// TIA Portal V20 export
DATA_BLOCK "MotorStarterHMI"   // DB212
// stored: MemoryReserve 100
   VAR
      unitMotorstarter : Array[0.."NO_OF_UNITS"] of "typeEmMotorStarterInterface";
   END_VAR
BEGIN
   unitMotorstarter[0].EMmotorstarter[0].et200SpMotorstarterCurrent[0..1] := 0.0;
   unitMotorstarter[0].EMmotorstarter[1].et200SpMotorstarterCurrent[0..1] := 0.0;
   unitMotorstarter[0].EMmotorstarter[2].et200SpMotorstarterCurrent[0..1] := 0.0;
   unitMotorstarter[0].EMmotorstarter[3].et200SpMotorstarterCurrent[0..1] := 0.0;
   unitMotorstarter[0].EMmotorstarter[4].et200SpMotorstarterCurrent[0..1] := 0.0;
   unitMotorstarter[0].EMmotorstarter[5].et200SpMotorstarterCurrent[0..1] := 0.0;
   unitMotorstarter[0].EMmotorstarter[6].et200SpMotorstarterCurrent[0..1] := 0.0;
   unitMotorstarter[0].EMmotorstarter[7].et200SpMotorstarterCurrent[0..1] := 0.0;
   unitMotorstarter[0].EMmotorstarter[0].et200SpMotorstarterInputs[0..1].readyAutomatic := FALSE;
   unitMotorstarter[0].EMmotorstarter[1].et200SpMotorstarterInputs[0..1].readyAutomatic := FALSE;
   unitMotorstarter[0].EMmotorstarter[2].et200SpMotorstarterInputs[0..1].readyAutomatic := FALSE;
   unitMotorstarter[0].EMmotorstarter[3].et200SpMotorstarterInputs[0..1].readyAutomatic := FALSE;
   unitMotorstarter[0].EMmotorstarter[4].et200SpMotorstarterInputs[0..1].readyAutomatic := FALSE;
   unitMotorstarter[0].EMmotorstarter[5].et200SpMotorstarterInputs[0..1].readyAutomatic := FALSE;
   unitMotorstarter[0].EMmotorstarter[6].et200SpMotorstarterInputs[0..1].readyAutomatic := FALSE;
   unitMotorstarter[0].EMmotorstarter[7].et200SpMotorstarterInputs[0..1].readyAutomatic := FALSE;
   unitMotorstarter[0].EMmotorstarter[0].et200SpMotorstarterInputs[0..1].motorOn := FALSE;
   unitMotorstarter[0].EMmotorstarter[1].et200SpMotorstarterInputs[0..1].motorOn := FALSE;
   unitMotorstarter[0].EMmotorstarter[2].et200SpMotorstarterInputs[0..1].motorOn := FALSE;
   unitMotorstarter[0].EMmotorstarter[3].et200SpMotorstarterInputs[0..1].motorOn := FALSE;
   unitMotorstarter[0].EMmotorstarter[4].et200SpMotorstarterInputs[0..1].motorOn := FALSE;
   unitMotorstarter[0].EMmotorstarter[5].et200SpMotorstarterInputs[0..1].motorOn := FALSE;
   unitMotorstarter[0].EMmotorstarter[6].et200SpMotorstarterInputs[0..1].motorOn := FALSE;
   unitMotorstarter[0].EMmotorstarter[7].et200SpMotorstarterInputs[0..1].motorOn := FALSE;
   unitMotorstarter[0].EMmotorstarter[0].et200SpMotorstarterInputs[0..1].groupFault := FALSE;
   unitMotorstarter[0].EMmotorstarter[1].et200SpMotorstarterInputs[0..1].groupFault := FALSE;
   unitMotorstarter[0].EMmotorstarter[2].et200SpMotorstarterInputs[0..1].groupFault := FALSE;
   unitMotorstarter[0].EMmotorstarter[3].et200SpMotorstarterInputs[0..1].groupFault := FALSE;
   unitMotorstarter[0].EMmotorstarter[4].et200SpMotorstarterInputs[0..1].groupFault := FALSE;
   unitMotorstarter[0].EMmotorstarter[5].et200SpMotorstarterInputs[0..1].groupFault := FALSE;
   unitMotorstarter[0].EMmotorstarter[6].et200SpMotorstarterInputs[0..1].groupFault := FALSE;
   unitMotorstarter[0].EMmotorstarter[7].et200SpMotorstarterInputs[0..1].groupFault := FALSE;
   unitMotorstarter[0].EMmotorstarter[0].et200SpMotorstarterInputs[0..1].groupWarning := FALSE;
   unitMotorstarter[0].EMmotorstarter[1].et200SpMotorstarterInputs[0..1].groupWarning := FALSE;
   unitMotorstarter[0].EMmotorstarter[2].et200SpMotorstarterInputs[0..1].groupWarning := FALSE;
   unitMotorstarter[0].EMmotorstarter[3].et200SpMotorstarterInputs[0..1].groupWarning := FALSE;
   unitMotorstarter[0].EMmotorstarter[4].et200SpMotorstarterInputs[0..1].groupWarning := FALSE;
   unitMotorstarter[0].EMmotorstarter[5].et200SpMotorstarterInputs[0..1].groupWarning := FALSE;
   unitMotorstarter[0].EMmotorstarter[6].et200SpMotorstarterInputs[0..1].groupWarning := FALSE;
   unitMotorstarter[0].EMmotorstarter[7].et200SpMotorstarterInputs[0..1].groupWarning := FALSE;
   unitMotorstarter[0].EMmotorstarter[0].et200SpMotorstarterInputs[0..1].input1 := FALSE;
   unitMotorstarter[0].EMmotorstarter[1].et200SpMotorstarterInputs[0..1].input1 := FALSE;
   unitMotorstarter[0].EMmotorstarter[2].et200SpMotorstarterInputs[0..1].input1 := FALSE;
   unitMotorstarter[0].EMmotorstarter[3].et200SpMotorstarterInputs[0..1].input1 := FALSE;
   unitMotorstarter[0].EMmotorstarter[4].et200SpMotorstarterInputs[0..1].input1 := FALSE;
   unitMotorstarter[0].EMmotorstarter[5].et200SpMotorstarterInputs[0..1].input1 := FALSE;
   unitMotorstarter[0].EMmotorstarter[6].et200SpMotorstarterInputs[0..1].input1 := FALSE;
   unitMotorstarter[0].EMmotorstarter[7].et200SpMotorstarterInputs[0..1].input1 := FALSE;
   unitMotorstarter[0].EMmotorstarter[0].et200SpMotorstarterInputs[0..1].input2 := FALSE;
   unitMotorstarter[0].EMmotorstarter[1].et200SpMotorstarterInputs[0..1].input2 := FALSE;
   unitMotorstarter[0].EMmotorstarter[2].et200SpMotorstarterInputs[0..1].input2 := FALSE;
   unitMotorstarter[0].EMmotorstarter[3].et200SpMotorstarterInputs[0..1].input2 := FALSE;
   unitMotorstarter[0].EMmotorstarter[4].et200SpMotorstarterInputs[0..1].input2 := FALSE;
   unitMotorstarter[0].EMmotorstarter[5].et200SpMotorstarterInputs[0..1].input2 := FALSE;
   unitMotorstarter[0].EMmotorstarter[6].et200SpMotorstarterInputs[0..1].input2 := FALSE;
   unitMotorstarter[0].EMmotorstarter[7].et200SpMotorstarterInputs[0..1].input2 := FALSE;
   unitMotorstarter[0].EMmotorstarter[0].et200SpMotorstarterInputs[0..1].input3 := FALSE;
   unitMotorstarter[0].EMmotorstarter[1].et200SpMotorstarterInputs[0..1].input3 := FALSE;
   unitMotorstarter[0].EMmotorstarter[2].et200SpMotorstarterInputs[0..1].input3 := FALSE;
   unitMotorstarter[0].EMmotorstarter[3].et200SpMotorstarterInputs[0..1].input3 := FALSE;
   unitMotorstarter[0].EMmotorstarter[4].et200SpMotorstarterInputs[0..1].input3 := FALSE;
   unitMotorstarter[0].EMmotorstarter[5].et200SpMotorstarterInputs[0..1].input3 := FALSE;
   unitMotorstarter[0].EMmotorstarter[6].et200SpMotorstarterInputs[0..1].input3 := FALSE;
   unitMotorstarter[0].EMmotorstarter[7].et200SpMotorstarterInputs[0..1].input3 := FALSE;
   unitMotorstarter[0].EMmotorstarter[0].et200SpMotorstarterInputs[0..1].inputLocalCtrl := FALSE;
   unitMotorstarter[0].EMmotorstarter[1].et200SpMotorstarterInputs[0..1].inputLocalCtrl := FALSE;
   unitMotorstarter[0].EMmotorstarter[2].et200SpMotorstarterInputs[0..1].inputLocalCtrl := FALSE;
   unitMotorstarter[0].EMmotorstarter[3].et200SpMotorstarterInputs[0..1].inputLocalCtrl := FALSE;
   unitMotorstarter[0].EMmotorstarter[4].et200SpMotorstarterInputs[0..1].inputLocalCtrl := FALSE;
   unitMotorstarter[0].EMmotorstarter[5].et200SpMotorstarterInputs[0..1].inputLocalCtrl := FALSE;
   unitMotorstarter[0].EMmotorstarter[6].et200SpMotorstarterInputs[0..1].inputLocalCtrl := FALSE;
   unitMotorstarter[0].EMmotorstarter[7].et200SpMotorstarterInputs[0..1].inputLocalCtrl := FALSE;
   unitMotorstarter[0].EMmotorstarter[0].et200SpMotorstarterInputs[0..1].iActBit0 := FALSE;
   unitMotorstarter[0].EMmotorstarter[1].et200SpMotorstarterInputs[0..1].iActBit0 := FALSE;
   unitMotorstarter[0].EMmotorstarter[2].et200SpMotorstarterInputs[0..1].iActBit0 := FALSE;
   unitMotorstarter[0].EMmotorstarter[3].et200SpMotorstarterInputs[0..1].iActBit0 := FALSE;
   unitMotorstarter[0].EMmotorstarter[4].et200SpMotorstarterInputs[0..1].iActBit0 := FALSE;
   unitMotorstarter[0].EMmotorstarter[5].et200SpMotorstarterInputs[0..1].iActBit0 := FALSE;
   unitMotorstarter[0].EMmotorstarter[6].et200SpMotorstarterInputs[0..1].iActBit0 := FALSE;
   unitMotorstarter[0].EMmotorstarter[7].et200SpMotorstarterInputs[0..1].iActBit0 := FALSE;
   unitMotorstarter[0].EMmotorstarter[0].et200SpMotorstarterInputs[0..1].iActBit1 := FALSE;
   unitMotorstarter[0].EMmotorstarter[1].et200SpMotorstarterInputs[0..1].iActBit1 := FALSE;
   unitMotorstarter[0].EMmotorstarter[2].et200SpMotorstarterInputs[0..1].iActBit1 := FALSE;
   unitMotorstarter[0].EMmotorstarter[3].et200SpMotorstarterInputs[0..1].iActBit1 := FALSE;
   unitMotorstarter[0].EMmotorstarter[4].et200SpMotorstarterInputs[0..1].iActBit1 := FALSE;
   unitMotorstarter[0].EMmotorstarter[5].et200SpMotorstarterInputs[0..1].iActBit1 := FALSE;
   unitMotorstarter[0].EMmotorstarter[6].et200SpMotorstarterInputs[0..1].iActBit1 := FALSE;
   unitMotorstarter[0].EMmotorstarter[7].et200SpMotorstarterInputs[0..1].iActBit1 := FALSE;
   unitMotorstarter[0].EMmotorstarter[0].et200SpMotorstarterInputs[0..1].iActBit2 := FALSE;
   unitMotorstarter[0].EMmotorstarter[1].et200SpMotorstarterInputs[0..1].iActBit2 := FALSE;
   unitMotorstarter[0].EMmotorstarter[2].et200SpMotorstarterInputs[0..1].iActBit2 := FALSE;
   unitMotorstarter[0].EMmotorstarter[3].et200SpMotorstarterInputs[0..1].iActBit2 := FALSE;
   unitMotorstarter[0].EMmotorstarter[4].et200SpMotorstarterInputs[0..1].iActBit2 := FALSE;
   unitMotorstarter[0].EMmotorstarter[5].et200SpMotorstarterInputs[0..1].iActBit2 := FALSE;
   unitMotorstarter[0].EMmotorstarter[6].et200SpMotorstarterInputs[0..1].iActBit2 := FALSE;
   unitMotorstarter[0].EMmotorstarter[7].et200SpMotorstarterInputs[0..1].iActBit2 := FALSE;
   unitMotorstarter[0].EMmotorstarter[0].et200SpMotorstarterInputs[0..1].iActBit3 := FALSE;
   unitMotorstarter[0].EMmotorstarter[1].et200SpMotorstarterInputs[0..1].iActBit3 := FALSE;
   unitMotorstarter[0].EMmotorstarter[2].et200SpMotorstarterInputs[0..1].iActBit3 := FALSE;
   unitMotorstarter[0].EMmotorstarter[3].et200SpMotorstarterInputs[0..1].iActBit3 := FALSE;
   unitMotorstarter[0].EMmotorstarter[4].et200SpMotorstarterInputs[0..1].iActBit3 := FALSE;
   unitMotorstarter[0].EMmotorstarter[5].et200SpMotorstarterInputs[0..1].iActBit3 := FALSE;
   unitMotorstarter[0].EMmotorstarter[6].et200SpMotorstarterInputs[0..1].iActBit3 := FALSE;
   unitMotorstarter[0].EMmotorstarter[7].et200SpMotorstarterInputs[0..1].iActBit3 := FALSE;
   unitMotorstarter[0].EMmotorstarter[0].et200SpMotorstarterInputs[0..1].iActBit4 := FALSE;
   unitMotorstarter[0].EMmotorstarter[1].et200SpMotorstarterInputs[0..1].iActBit4 := FALSE;
   unitMotorstarter[0].EMmotorstarter[2].et200SpMotorstarterInputs[0..1].iActBit4 := FALSE;
   unitMotorstarter[0].EMmotorstarter[3].et200SpMotorstarterInputs[0..1].iActBit4 := FALSE;
   unitMotorstarter[0].EMmotorstarter[4].et200SpMotorstarterInputs[0..1].iActBit4 := FALSE;
   unitMotorstarter[0].EMmotorstarter[5].et200SpMotorstarterInputs[0..1].iActBit4 := FALSE;
   unitMotorstarter[0].EMmotorstarter[6].et200SpMotorstarterInputs[0..1].iActBit4 := FALSE;
   unitMotorstarter[0].EMmotorstarter[7].et200SpMotorstarterInputs[0..1].iActBit4 := FALSE;
   unitMotorstarter[0].EMmotorstarter[0].et200SpMotorstarterInputs[0..1].iActBit5 := FALSE;
   unitMotorstarter[0].EMmotorstarter[1].et200SpMotorstarterInputs[0..1].iActBit5 := FALSE;
   unitMotorstarter[0].EMmotorstarter[2].et200SpMotorstarterInputs[0..1].iActBit5 := FALSE;
   unitMotorstarter[0].EMmotorstarter[3].et200SpMotorstarterInputs[0..1].iActBit5 := FALSE;
   unitMotorstarter[0].EMmotorstarter[4].et200SpMotorstarterInputs[0..1].iActBit5 := FALSE;
   unitMotorstarter[0].EMmotorstarter[5].et200SpMotorstarterInputs[0..1].iActBit5 := FALSE;
   unitMotorstarter[0].EMmotorstarter[6].et200SpMotorstarterInputs[0..1].iActBit5 := FALSE;
   unitMotorstarter[0].EMmotorstarter[7].et200SpMotorstarterInputs[0..1].iActBit5 := FALSE;
   unitMotorstarter[0].EMmotorstarter[0].et200SpMotorstarterInputs[0..1].manualOperating := FALSE;
   unitMotorstarter[0].EMmotorstarter[1].et200SpMotorstarterInputs[0..1].manualOperating := FALSE;
   unitMotorstarter[0].EMmotorstarter[2].et200SpMotorstarterInputs[0..1].manualOperating := FALSE;
   unitMotorstarter[0].EMmotorstarter[3].et200SpMotorstarterInputs[0..1].manualOperating := FALSE;
   unitMotorstarter[0].EMmotorstarter[4].et200SpMotorstarterInputs[0..1].manualOperating := FALSE;
   unitMotorstarter[0].EMmotorstarter[5].et200SpMotorstarterInputs[0..1].manualOperating := FALSE;
   unitMotorstarter[0].EMmotorstarter[6].et200SpMotorstarterInputs[0..1].manualOperating := FALSE;
   unitMotorstarter[0].EMmotorstarter[7].et200SpMotorstarterInputs[0..1].manualOperating := FALSE;
   unitMotorstarter[0].EMmotorstarter[0].et200SpMotorstarterInputs[0..1].spare1 := FALSE;
   unitMotorstarter[0].EMmotorstarter[1].et200SpMotorstarterInputs[0..1].spare1 := FALSE;
   unitMotorstarter[0].EMmotorstarter[2].et200SpMotorstarterInputs[0..1].spare1 := FALSE;
   unitMotorstarter[0].EMmotorstarter[3].et200SpMotorstarterInputs[0..1].spare1 := FALSE;
   unitMotorstarter[0].EMmotorstarter[4].et200SpMotorstarterInputs[0..1].spare1 := FALSE;
   unitMotorstarter[0].EMmotorstarter[5].et200SpMotorstarterInputs[0..1].spare1 := FALSE;
   unitMotorstarter[0].EMmotorstarter[6].et200SpMotorstarterInputs[0..1].spare1 := FALSE;
   unitMotorstarter[0].EMmotorstarter[7].et200SpMotorstarterInputs[0..1].spare1 := FALSE;
   unitMotorstarter[0].EMmotorstarter[0].et200SpMotorstarterInputs[0..1].readyStartOn := FALSE;
   unitMotorstarter[0].EMmotorstarter[1].et200SpMotorstarterInputs[0..1].readyStartOn := FALSE;
   unitMotorstarter[0].EMmotorstarter[2].et200SpMotorstarterInputs[0..1].readyStartOn := FALSE;
   unitMotorstarter[0].EMmotorstarter[3].et200SpMotorstarterInputs[0..1].readyStartOn := FALSE;
   unitMotorstarter[0].EMmotorstarter[4].et200SpMotorstarterInputs[0..1].readyStartOn := FALSE;
   unitMotorstarter[0].EMmotorstarter[5].et200SpMotorstarterInputs[0..1].readyStartOn := FALSE;
   unitMotorstarter[0].EMmotorstarter[6].et200SpMotorstarterInputs[0..1].readyStartOn := FALSE;
   unitMotorstarter[0].EMmotorstarter[7].et200SpMotorstarterInputs[0..1].readyStartOn := FALSE;
   unitMotorstarter[0].EMmotorstarter[0].et200SpMotorstarterInputs[0..1].motorOnRight := FALSE;
   unitMotorstarter[0].EMmotorstarter[1].et200SpMotorstarterInputs[0..1].motorOnRight := FALSE;
   unitMotorstarter[0].EMmotorstarter[2].et200SpMotorstarterInputs[0..1].motorOnRight := FALSE;
   unitMotorstarter[0].EMmotorstarter[3].et200SpMotorstarterInputs[0..1].motorOnRight := FALSE;
   unitMotorstarter[0].EMmotorstarter[4].et200SpMotorstarterInputs[0..1].motorOnRight := FALSE;
   unitMotorstarter[0].EMmotorstarter[5].et200SpMotorstarterInputs[0..1].motorOnRight := FALSE;
   unitMotorstarter[0].EMmotorstarter[6].et200SpMotorstarterInputs[0..1].motorOnRight := FALSE;
   unitMotorstarter[0].EMmotorstarter[7].et200SpMotorstarterInputs[0..1].motorOnRight := FALSE;
   unitMotorstarter[0].EMmotorstarter[0].et200SpMotorstarterInputs[0..1].motorOnLeft := FALSE;
   unitMotorstarter[0].EMmotorstarter[1].et200SpMotorstarterInputs[0..1].motorOnLeft := FALSE;
   unitMotorstarter[0].EMmotorstarter[2].et200SpMotorstarterInputs[0..1].motorOnLeft := FALSE;
   unitMotorstarter[0].EMmotorstarter[3].et200SpMotorstarterInputs[0..1].motorOnLeft := FALSE;
   unitMotorstarter[0].EMmotorstarter[4].et200SpMotorstarterInputs[0..1].motorOnLeft := FALSE;
   unitMotorstarter[0].EMmotorstarter[5].et200SpMotorstarterInputs[0..1].motorOnLeft := FALSE;
   unitMotorstarter[0].EMmotorstarter[6].et200SpMotorstarterInputs[0..1].motorOnLeft := FALSE;
   unitMotorstarter[0].EMmotorstarter[7].et200SpMotorstarterInputs[0..1].motorOnLeft := FALSE;
   unitMotorstarter[0].EMmotorstarter[0].et200SpMotorstarterInputs[0..1].quickstopActive := FALSE;
   unitMotorstarter[0].EMmotorstarter[1].et200SpMotorstarterInputs[0..1].quickstopActive := FALSE;
   unitMotorstarter[0].EMmotorstarter[2].et200SpMotorstarterInputs[0..1].quickstopActive := FALSE;
   unitMotorstarter[0].EMmotorstarter[3].et200SpMotorstarterInputs[0..1].quickstopActive := FALSE;
   unitMotorstarter[0].EMmotorstarter[4].et200SpMotorstarterInputs[0..1].quickstopActive := FALSE;
   unitMotorstarter[0].EMmotorstarter[5].et200SpMotorstarterInputs[0..1].quickstopActive := FALSE;
   unitMotorstarter[0].EMmotorstarter[6].et200SpMotorstarterInputs[0..1].quickstopActive := FALSE;
   unitMotorstarter[0].EMmotorstarter[7].et200SpMotorstarterInputs[0..1].quickstopActive := FALSE;
   unitMotorstarter[0].EMmotorstarter[0].et200SpMotorstarterInputs[0..1].energySaving := FALSE;
   unitMotorstarter[0].EMmotorstarter[1].et200SpMotorstarterInputs[0..1].energySaving := FALSE;
   unitMotorstarter[0].EMmotorstarter[2].et200SpMotorstarterInputs[0..1].energySaving := FALSE;
   unitMotorstarter[0].EMmotorstarter[3].et200SpMotorstarterInputs[0..1].energySaving := FALSE;
   unitMotorstarter[0].EMmotorstarter[4].et200SpMotorstarterInputs[0..1].energySaving := FALSE;
   unitMotorstarter[0].EMmotorstarter[5].et200SpMotorstarterInputs[0..1].energySaving := FALSE;
   unitMotorstarter[0].EMmotorstarter[6].et200SpMotorstarterInputs[0..1].energySaving := FALSE;
   unitMotorstarter[0].EMmotorstarter[7].et200SpMotorstarterInputs[0..1].energySaving := FALSE;
   unitMotorstarter[0].EMmotorstarter[0].et200SpMotorstarterInputs[0..1].moduleInserted := FALSE;
   unitMotorstarter[0].EMmotorstarter[1].et200SpMotorstarterInputs[0..1].moduleInserted := FALSE;
   unitMotorstarter[0].EMmotorstarter[2].et200SpMotorstarterInputs[0..1].moduleInserted := FALSE;
   unitMotorstarter[0].EMmotorstarter[3].et200SpMotorstarterInputs[0..1].moduleInserted := FALSE;
   unitMotorstarter[0].EMmotorstarter[4].et200SpMotorstarterInputs[0..1].moduleInserted := FALSE;
   unitMotorstarter[0].EMmotorstarter[5].et200SpMotorstarterInputs[0..1].moduleInserted := FALSE;
   unitMotorstarter[0].EMmotorstarter[6].et200SpMotorstarterInputs[0..1].moduleInserted := FALSE;
   unitMotorstarter[0].EMmotorstarter[7].et200SpMotorstarterInputs[0..1].moduleInserted := FALSE;
   unitMotorstarter[0].EMmotorstarter[0].et200SpMotorstarterInputs[0..1].exProtectionMotorActive := FALSE;
   unitMotorstarter[0].EMmotorstarter[1].et200SpMotorstarterInputs[0..1].exProtectionMotorActive := FALSE;
   unitMotorstarter[0].EMmotorstarter[2].et200SpMotorstarterInputs[0..1].exProtectionMotorActive := FALSE;
   unitMotorstarter[0].EMmotorstarter[3].et200SpMotorstarterInputs[0..1].exProtectionMotorActive := FALSE;
   unitMotorstarter[0].EMmotorstarter[4].et200SpMotorstarterInputs[0..1].exProtectionMotorActive := FALSE;
   unitMotorstarter[0].EMmotorstarter[5].et200SpMotorstarterInputs[0..1].exProtectionMotorActive := FALSE;
   unitMotorstarter[0].EMmotorstarter[6].et200SpMotorstarterInputs[0..1].exProtectionMotorActive := FALSE;
   unitMotorstarter[0].EMmotorstarter[7].et200SpMotorstarterInputs[0..1].exProtectionMotorActive := FALSE;
   unitMotorstarter[0].EMmotorstarter[0].et200SpMotorstarterInputs[0..1].blockActive := FALSE;
   unitMotorstarter[0].EMmotorstarter[1].et200SpMotorstarterInputs[0..1].blockActive := FALSE;
   unitMotorstarter[0].EMmotorstarter[2].et200SpMotorstarterInputs[0..1].blockActive := FALSE;
   unitMotorstarter[0].EMmotorstarter[3].et200SpMotorstarterInputs[0..1].blockActive := FALSE;
   unitMotorstarter[0].EMmotorstarter[4].et200SpMotorstarterInputs[0..1].blockActive := FALSE;
   unitMotorstarter[0].EMmotorstarter[5].et200SpMotorstarterInputs[0..1].blockActive := FALSE;
   unitMotorstarter[0].EMmotorstarter[6].et200SpMotorstarterInputs[0..1].blockActive := FALSE;
   unitMotorstarter[0].EMmotorstarter[7].et200SpMotorstarterInputs[0..1].blockActive := FALSE;
   unitMotorstarter[0].EMmotorstarter[0].et200SpMotorstarterInputs[0..1].thermalMotorOverload := FALSE;
   unitMotorstarter[0].EMmotorstarter[1].et200SpMotorstarterInputs[0..1].thermalMotorOverload := FALSE;
   unitMotorstarter[0].EMmotorstarter[2].et200SpMotorstarterInputs[0..1].thermalMotorOverload := FALSE;
   unitMotorstarter[0].EMmotorstarter[3].et200SpMotorstarterInputs[0..1].thermalMotorOverload := FALSE;
   unitMotorstarter[0].EMmotorstarter[4].et200SpMotorstarterInputs[0..1].thermalMotorOverload := FALSE;
   unitMotorstarter[0].EMmotorstarter[5].et200SpMotorstarterInputs[0..1].thermalMotorOverload := FALSE;
   unitMotorstarter[0].EMmotorstarter[6].et200SpMotorstarterInputs[0..1].thermalMotorOverload := FALSE;
   unitMotorstarter[0].EMmotorstarter[7].et200SpMotorstarterInputs[0..1].thermalMotorOverload := FALSE;
   unitMotorstarter[0].EMmotorstarter[0].et200SpMotorstarterInputs[0..1].spare5 := FALSE;
   unitMotorstarter[0].EMmotorstarter[1].et200SpMotorstarterInputs[0..1].spare5 := FALSE;
   unitMotorstarter[0].EMmotorstarter[2].et200SpMotorstarterInputs[0..1].spare5 := FALSE;
   unitMotorstarter[0].EMmotorstarter[3].et200SpMotorstarterInputs[0..1].spare5 := FALSE;
   unitMotorstarter[0].EMmotorstarter[4].et200SpMotorstarterInputs[0..1].spare5 := FALSE;
   unitMotorstarter[0].EMmotorstarter[5].et200SpMotorstarterInputs[0..1].spare5 := FALSE;
   unitMotorstarter[0].EMmotorstarter[6].et200SpMotorstarterInputs[0..1].spare5 := FALSE;
   unitMotorstarter[0].EMmotorstarter[7].et200SpMotorstarterInputs[0..1].spare5 := FALSE;
   unitMotorstarter[0].EMmotorstarter[0].et200SpMotorstarterInputs[0..1].currentLimitTripping := FALSE;
   unitMotorstarter[0].EMmotorstarter[1].et200SpMotorstarterInputs[0..1].currentLimitTripping := FALSE;
   unitMotorstarter[0].EMmotorstarter[2].et200SpMotorstarterInputs[0..1].currentLimitTripping := FALSE;
   unitMotorstarter[0].EMmotorstarter[3].et200SpMotorstarterInputs[0..1].currentLimitTripping := FALSE;
   unitMotorstarter[0].EMmotorstarter[4].et200SpMotorstarterInputs[0..1].currentLimitTripping := FALSE;
   unitMotorstarter[0].EMmotorstarter[5].et200SpMotorstarterInputs[0..1].currentLimitTripping := FALSE;
   unitMotorstarter[0].EMmotorstarter[6].et200SpMotorstarterInputs[0..1].currentLimitTripping := FALSE;
   unitMotorstarter[0].EMmotorstarter[7].et200SpMotorstarterInputs[0..1].currentLimitTripping := FALSE;
   unitMotorstarter[0].EMmotorstarter[0].et200SpMotorstarterInputs[0..1].statusFailDi := FALSE;
   unitMotorstarter[0].EMmotorstarter[1].et200SpMotorstarterInputs[0..1].statusFailDi := FALSE;
   unitMotorstarter[0].EMmotorstarter[2].et200SpMotorstarterInputs[0..1].statusFailDi := FALSE;
   unitMotorstarter[0].EMmotorstarter[3].et200SpMotorstarterInputs[0..1].statusFailDi := FALSE;
   unitMotorstarter[0].EMmotorstarter[4].et200SpMotorstarterInputs[0..1].statusFailDi := FALSE;
   unitMotorstarter[0].EMmotorstarter[5].et200SpMotorstarterInputs[0..1].statusFailDi := FALSE;
   unitMotorstarter[0].EMmotorstarter[6].et200SpMotorstarterInputs[0..1].statusFailDi := FALSE;
   unitMotorstarter[0].EMmotorstarter[7].et200SpMotorstarterInputs[0..1].statusFailDi := FALSE;
   unitMotorstarter[0].EMmotorstarter[0].et200SpMotorstarterInputs[0..1].residualCurrent := FALSE;
   unitMotorstarter[0].EMmotorstarter[1].et200SpMotorstarterInputs[0..1].residualCurrent := FALSE;
   unitMotorstarter[0].EMmotorstarter[2].et200SpMotorstarterInputs[0..1].residualCurrent := FALSE;
   unitMotorstarter[0].EMmotorstarter[3].et200SpMotorstarterInputs[0..1].residualCurrent := FALSE;
   unitMotorstarter[0].EMmotorstarter[4].et200SpMotorstarterInputs[0..1].residualCurrent := FALSE;
   unitMotorstarter[0].EMmotorstarter[5].et200SpMotorstarterInputs[0..1].residualCurrent := FALSE;
   unitMotorstarter[0].EMmotorstarter[6].et200SpMotorstarterInputs[0..1].residualCurrent := FALSE;
   unitMotorstarter[0].EMmotorstarter[7].et200SpMotorstarterInputs[0..1].residualCurrent := FALSE;
   unitMotorstarter[0].EMmotorstarter[0].et200SpMotorstarterInputs[0..1].asymmetryDetected := FALSE;
   unitMotorstarter[0].EMmotorstarter[1].et200SpMotorstarterInputs[0..1].asymmetryDetected := FALSE;
   unitMotorstarter[0].EMmotorstarter[2].et200SpMotorstarterInputs[0..1].asymmetryDetected := FALSE;
   unitMotorstarter[0].EMmotorstarter[3].et200SpMotorstarterInputs[0..1].asymmetryDetected := FALSE;
   unitMotorstarter[0].EMmotorstarter[4].et200SpMotorstarterInputs[0..1].asymmetryDetected := FALSE;
   unitMotorstarter[0].EMmotorstarter[5].et200SpMotorstarterInputs[0..1].asymmetryDetected := FALSE;
   unitMotorstarter[0].EMmotorstarter[6].et200SpMotorstarterInputs[0..1].asymmetryDetected := FALSE;
   unitMotorstarter[0].EMmotorstarter[7].et200SpMotorstarterInputs[0..1].asymmetryDetected := FALSE;
   unitMotorstarter[0].EMmotorstarter[0].et200SpMotorstarterInputs[0..1].overtemperature := FALSE;
   unitMotorstarter[0].EMmotorstarter[1].et200SpMotorstarterInputs[0..1].overtemperature := FALSE;
   unitMotorstarter[0].EMmotorstarter[2].et200SpMotorstarterInputs[0..1].overtemperature := FALSE;
   unitMotorstarter[0].EMmotorstarter[3].et200SpMotorstarterInputs[0..1].overtemperature := FALSE;
   unitMotorstarter[0].EMmotorstarter[4].et200SpMotorstarterInputs[0..1].overtemperature := FALSE;
   unitMotorstarter[0].EMmotorstarter[5].et200SpMotorstarterInputs[0..1].overtemperature := FALSE;
   unitMotorstarter[0].EMmotorstarter[6].et200SpMotorstarterInputs[0..1].overtemperature := FALSE;
   unitMotorstarter[0].EMmotorstarter[7].et200SpMotorstarterInputs[0..1].overtemperature := FALSE;
   unitMotorstarter[0].EMmotorstarter[0].et200SpMotorstarterInputs[0..1].spare7 := FALSE;
   unitMotorstarter[0].EMmotorstarter[1].et200SpMotorstarterInputs[0..1].spare7 := FALSE;
   unitMotorstarter[0].EMmotorstarter[2].et200SpMotorstarterInputs[0..1].spare7 := FALSE;
   unitMotorstarter[0].EMmotorstarter[3].et200SpMotorstarterInputs[0..1].spare7 := FALSE;
   unitMotorstarter[0].EMmotorstarter[4].et200SpMotorstarterInputs[0..1].spare7 := FALSE;
   unitMotorstarter[0].EMmotorstarter[5].et200SpMotorstarterInputs[0..1].spare7 := FALSE;
   unitMotorstarter[0].EMmotorstarter[6].et200SpMotorstarterInputs[0..1].spare7 := FALSE;
   unitMotorstarter[0].EMmotorstarter[7].et200SpMotorstarterInputs[0..1].spare7 := FALSE;
   unitMotorstarter[0].EMmotorstarter[0].et200SpMotorstarterOutputs[0..1].motorCw := FALSE;
   unitMotorstarter[0].EMmotorstarter[1].et200SpMotorstarterOutputs[0..1].motorCw := FALSE;
   unitMotorstarter[0].EMmotorstarter[2].et200SpMotorstarterOutputs[0..1].motorCw := FALSE;
   unitMotorstarter[0].EMmotorstarter[3].et200SpMotorstarterOutputs[0..1].motorCw := FALSE;
   unitMotorstarter[0].EMmotorstarter[4].et200SpMotorstarterOutputs[0..1].motorCw := FALSE;
   unitMotorstarter[0].EMmotorstarter[5].et200SpMotorstarterOutputs[0..1].motorCw := FALSE;
   unitMotorstarter[0].EMmotorstarter[6].et200SpMotorstarterOutputs[0..1].motorCw := FALSE;
   unitMotorstarter[0].EMmotorstarter[7].et200SpMotorstarterOutputs[0..1].motorCw := FALSE;
   unitMotorstarter[0].EMmotorstarter[0].et200SpMotorstarterOutputs[0..1].motorCww := FALSE;
   unitMotorstarter[0].EMmotorstarter[1].et200SpMotorstarterOutputs[0..1].motorCww := FALSE;
   unitMotorstarter[0].EMmotorstarter[2].et200SpMotorstarterOutputs[0..1].motorCww := FALSE;
   unitMotorstarter[0].EMmotorstarter[3].et200SpMotorstarterOutputs[0..1].motorCww := FALSE;
   unitMotorstarter[0].EMmotorstarter[4].et200SpMotorstarterOutputs[0..1].motorCww := FALSE;
   unitMotorstarter[0].EMmotorstarter[5].et200SpMotorstarterOutputs[0..1].motorCww := FALSE;
   unitMotorstarter[0].EMmotorstarter[6].et200SpMotorstarterOutputs[0..1].motorCww := FALSE;
   unitMotorstarter[0].EMmotorstarter[7].et200SpMotorstarterOutputs[0..1].motorCww := FALSE;
   unitMotorstarter[0].EMmotorstarter[0].et200SpMotorstarterOutputs[0..1].reserve1 := FALSE;
   unitMotorstarter[0].EMmotorstarter[1].et200SpMotorstarterOutputs[0..1].reserve1 := FALSE;
   unitMotorstarter[0].EMmotorstarter[2].et200SpMotorstarterOutputs[0..1].reserve1 := FALSE;
   unitMotorstarter[0].EMmotorstarter[3].et200SpMotorstarterOutputs[0..1].reserve1 := FALSE;
   unitMotorstarter[0].EMmotorstarter[4].et200SpMotorstarterOutputs[0..1].reserve1 := FALSE;
   unitMotorstarter[0].EMmotorstarter[5].et200SpMotorstarterOutputs[0..1].reserve1 := FALSE;
   unitMotorstarter[0].EMmotorstarter[6].et200SpMotorstarterOutputs[0..1].reserve1 := FALSE;
   unitMotorstarter[0].EMmotorstarter[7].et200SpMotorstarterOutputs[0..1].reserve1 := FALSE;
   unitMotorstarter[0].EMmotorstarter[0].et200SpMotorstarterOutputs[0..1].tripReset := FALSE;
   unitMotorstarter[0].EMmotorstarter[1].et200SpMotorstarterOutputs[0..1].tripReset := FALSE;
   unitMotorstarter[0].EMmotorstarter[2].et200SpMotorstarterOutputs[0..1].tripReset := FALSE;
   unitMotorstarter[0].EMmotorstarter[3].et200SpMotorstarterOutputs[0..1].tripReset := FALSE;
   unitMotorstarter[0].EMmotorstarter[4].et200SpMotorstarterOutputs[0..1].tripReset := FALSE;
   unitMotorstarter[0].EMmotorstarter[5].et200SpMotorstarterOutputs[0..1].tripReset := FALSE;
   unitMotorstarter[0].EMmotorstarter[6].et200SpMotorstarterOutputs[0..1].tripReset := FALSE;
   unitMotorstarter[0].EMmotorstarter[7].et200SpMotorstarterOutputs[0..1].tripReset := FALSE;
   unitMotorstarter[0].EMmotorstarter[0].et200SpMotorstarterOutputs[0..1].emergencyStart := FALSE;
   unitMotorstarter[0].EMmotorstarter[1].et200SpMotorstarterOutputs[0..1].emergencyStart := FALSE;
   unitMotorstarter[0].EMmotorstarter[2].et200SpMotorstarterOutputs[0..1].emergencyStart := FALSE;
   unitMotorstarter[0].EMmotorstarter[3].et200SpMotorstarterOutputs[0..1].emergencyStart := FALSE;
   unitMotorstarter[0].EMmotorstarter[4].et200SpMotorstarterOutputs[0..1].emergencyStart := FALSE;
   unitMotorstarter[0].EMmotorstarter[5].et200SpMotorstarterOutputs[0..1].emergencyStart := FALSE;
   unitMotorstarter[0].EMmotorstarter[6].et200SpMotorstarterOutputs[0..1].emergencyStart := FALSE;
   unitMotorstarter[0].EMmotorstarter[7].et200SpMotorstarterOutputs[0..1].emergencyStart := FALSE;
   unitMotorstarter[0].EMmotorstarter[0].et200SpMotorstarterOutputs[0..1].reserve2 := FALSE;
   unitMotorstarter[0].EMmotorstarter[1].et200SpMotorstarterOutputs[0..1].reserve2 := FALSE;
   unitMotorstarter[0].EMmotorstarter[2].et200SpMotorstarterOutputs[0..1].reserve2 := FALSE;
   unitMotorstarter[0].EMmotorstarter[3].et200SpMotorstarterOutputs[0..1].reserve2 := FALSE;
   unitMotorstarter[0].EMmotorstarter[4].et200SpMotorstarterOutputs[0..1].reserve2 := FALSE;
   unitMotorstarter[0].EMmotorstarter[5].et200SpMotorstarterOutputs[0..1].reserve2 := FALSE;
   unitMotorstarter[0].EMmotorstarter[6].et200SpMotorstarterOutputs[0..1].reserve2 := FALSE;
   unitMotorstarter[0].EMmotorstarter[7].et200SpMotorstarterOutputs[0..1].reserve2 := FALSE;
   unitMotorstarter[0].EMmotorstarter[0].et200SpMotorstarterOutputs[0..1].reserve3 := FALSE;
   unitMotorstarter[0].EMmotorstarter[1].et200SpMotorstarterOutputs[0..1].reserve3 := FALSE;
   unitMotorstarter[0].EMmotorstarter[2].et200SpMotorstarterOutputs[0..1].reserve3 := FALSE;
   unitMotorstarter[0].EMmotorstarter[3].et200SpMotorstarterOutputs[0..1].reserve3 := FALSE;
   unitMotorstarter[0].EMmotorstarter[4].et200SpMotorstarterOutputs[0..1].reserve3 := FALSE;
   unitMotorstarter[0].EMmotorstarter[5].et200SpMotorstarterOutputs[0..1].reserve3 := FALSE;
   unitMotorstarter[0].EMmotorstarter[6].et200SpMotorstarterOutputs[0..1].reserve3 := FALSE;
   unitMotorstarter[0].EMmotorstarter[7].et200SpMotorstarterOutputs[0..1].reserve3 := FALSE;
   unitMotorstarter[0].EMmotorstarter[0].et200SpMotorstarterOutputs[0..1].coldStart := FALSE;
   unitMotorstarter[0].EMmotorstarter[1].et200SpMotorstarterOutputs[0..1].coldStart := FALSE;
   unitMotorstarter[0].EMmotorstarter[2].et200SpMotorstarterOutputs[0..1].coldStart := FALSE;
   unitMotorstarter[0].EMmotorstarter[3].et200SpMotorstarterOutputs[0..1].coldStart := FALSE;
   unitMotorstarter[0].EMmotorstarter[4].et200SpMotorstarterOutputs[0..1].coldStart := FALSE;
   unitMotorstarter[0].EMmotorstarter[5].et200SpMotorstarterOutputs[0..1].coldStart := FALSE;
   unitMotorstarter[0].EMmotorstarter[6].et200SpMotorstarterOutputs[0..1].coldStart := FALSE;
   unitMotorstarter[0].EMmotorstarter[7].et200SpMotorstarterOutputs[0..1].coldStart := FALSE;
   unitMotorstarter[0].EMmotorstarter[0].et200SpMotorstarterOutputs[0..1].reserve4 := FALSE;
   unitMotorstarter[0].EMmotorstarter[1].et200SpMotorstarterOutputs[0..1].reserve4 := FALSE;
   unitMotorstarter[0].EMmotorstarter[2].et200SpMotorstarterOutputs[0..1].reserve4 := FALSE;
   unitMotorstarter[0].EMmotorstarter[3].et200SpMotorstarterOutputs[0..1].reserve4 := FALSE;
   unitMotorstarter[0].EMmotorstarter[4].et200SpMotorstarterOutputs[0..1].reserve4 := FALSE;
   unitMotorstarter[0].EMmotorstarter[5].et200SpMotorstarterOutputs[0..1].reserve4 := FALSE;
   unitMotorstarter[0].EMmotorstarter[6].et200SpMotorstarterOutputs[0..1].reserve4 := FALSE;
   unitMotorstarter[0].EMmotorstarter[7].et200SpMotorstarterOutputs[0..1].reserve4 := FALSE;
   unitMotorstarter[0].EMmotorstarter[0].et200SpMotorstarterOutputs[0..1].reserve5 := FALSE;
   unitMotorstarter[0].EMmotorstarter[1].et200SpMotorstarterOutputs[0..1].reserve5 := FALSE;
   unitMotorstarter[0].EMmotorstarter[2].et200SpMotorstarterOutputs[0..1].reserve5 := FALSE;
   unitMotorstarter[0].EMmotorstarter[3].et200SpMotorstarterOutputs[0..1].reserve5 := FALSE;
   unitMotorstarter[0].EMmotorstarter[4].et200SpMotorstarterOutputs[0..1].reserve5 := FALSE;
   unitMotorstarter[0].EMmotorstarter[5].et200SpMotorstarterOutputs[0..1].reserve5 := FALSE;
   unitMotorstarter[0].EMmotorstarter[6].et200SpMotorstarterOutputs[0..1].reserve5 := FALSE;
   unitMotorstarter[0].EMmotorstarter[7].et200SpMotorstarterOutputs[0..1].reserve5 := FALSE;
   unitMotorstarter[0].EMmotorstarter[0].et200SpMotorstarterOutputs[0..1].reserve6 := FALSE;
   unitMotorstarter[0].EMmotorstarter[1].et200SpMotorstarterOutputs[0..1].reserve6 := FALSE;
   unitMotorstarter[0].EMmotorstarter[2].et200SpMotorstarterOutputs[0..1].reserve6 := FALSE;
   unitMotorstarter[0].EMmotorstarter[3].et200SpMotorstarterOutputs[0..1].reserve6 := FALSE;
   unitMotorstarter[0].EMmotorstarter[4].et200SpMotorstarterOutputs[0..1].reserve6 := FALSE;
   unitMotorstarter[0].EMmotorstarter[5].et200SpMotorstarterOutputs[0..1].reserve6 := FALSE;
   unitMotorstarter[0].EMmotorstarter[6].et200SpMotorstarterOutputs[0..1].reserve6 := FALSE;
   unitMotorstarter[0].EMmotorstarter[7].et200SpMotorstarterOutputs[0..1].reserve6 := FALSE;
   unitMotorstarter[0].EMmotorstarter[0].et200SpMotorstarterOutputs[0..1].reserve7 := FALSE;
   unitMotorstarter[0].EMmotorstarter[1].et200SpMotorstarterOutputs[0..1].reserve7 := FALSE;
   unitMotorstarter[0].EMmotorstarter[2].et200SpMotorstarterOutputs[0..1].reserve7 := FALSE;
   unitMotorstarter[0].EMmotorstarter[3].et200SpMotorstarterOutputs[0..1].reserve7 := FALSE;
   unitMotorstarter[0].EMmotorstarter[4].et200SpMotorstarterOutputs[0..1].reserve7 := FALSE;
   unitMotorstarter[0].EMmotorstarter[5].et200SpMotorstarterOutputs[0..1].reserve7 := FALSE;
   unitMotorstarter[0].EMmotorstarter[6].et200SpMotorstarterOutputs[0..1].reserve7 := FALSE;
   unitMotorstarter[0].EMmotorstarter[7].et200SpMotorstarterOutputs[0..1].reserve7 := FALSE;
   unitMotorstarter[0].EMmotorstarter[0].et200SpMotorstarterOutputs[0..1].reserve8 := FALSE;
   unitMotorstarter[0].EMmotorstarter[1].et200SpMotorstarterOutputs[0..1].reserve8 := FALSE;
   unitMotorstarter[0].EMmotorstarter[2].et200SpMotorstarterOutputs[0..1].reserve8 := FALSE;
   unitMotorstarter[0].EMmotorstarter[3].et200SpMotorstarterOutputs[0..1].reserve8 := FALSE;
   unitMotorstarter[0].EMmotorstarter[4].et200SpMotorstarterOutputs[0..1].reserve8 := FALSE;
   unitMotorstarter[0].EMmotorstarter[5].et200SpMotorstarterOutputs[0..1].reserve8 := FALSE;
   unitMotorstarter[0].EMmotorstarter[6].et200SpMotorstarterOutputs[0..1].reserve8 := FALSE;
   unitMotorstarter[0].EMmotorstarter[7].et200SpMotorstarterOutputs[0..1].reserve8 := FALSE;
   unitMotorstarter[0].EMmotorstarter[0].et200SpMotorstarterOutputs[0..1].reserve9 := FALSE;
   unitMotorstarter[0].EMmotorstarter[1].et200SpMotorstarterOutputs[0..1].reserve9 := FALSE;
   unitMotorstarter[0].EMmotorstarter[2].et200SpMotorstarterOutputs[0..1].reserve9 := FALSE;
   unitMotorstarter[0].EMmotorstarter[3].et200SpMotorstarterOutputs[0..1].reserve9 := FALSE;
   unitMotorstarter[0].EMmotorstarter[4].et200SpMotorstarterOutputs[0..1].reserve9 := FALSE;
   unitMotorstarter[0].EMmotorstarter[5].et200SpMotorstarterOutputs[0..1].reserve9 := FALSE;
   unitMotorstarter[0].EMmotorstarter[6].et200SpMotorstarterOutputs[0..1].reserve9 := FALSE;
   unitMotorstarter[0].EMmotorstarter[7].et200SpMotorstarterOutputs[0..1].reserve9 := FALSE;
   unitMotorstarter[0].EMmotorstarter[0].et200SpMotorstarterOutputs[0..1].reserve10 := FALSE;
   unitMotorstarter[0].EMmotorstarter[1].et200SpMotorstarterOutputs[0..1].reserve10 := FALSE;
   unitMotorstarter[0].EMmotorstarter[2].et200SpMotorstarterOutputs[0..1].reserve10 := FALSE;
   unitMotorstarter[0].EMmotorstarter[3].et200SpMotorstarterOutputs[0..1].reserve10 := FALSE;
   unitMotorstarter[0].EMmotorstarter[4].et200SpMotorstarterOutputs[0..1].reserve10 := FALSE;
   unitMotorstarter[0].EMmotorstarter[5].et200SpMotorstarterOutputs[0..1].reserve10 := FALSE;
   unitMotorstarter[0].EMmotorstarter[6].et200SpMotorstarterOutputs[0..1].reserve10 := FALSE;
   unitMotorstarter[0].EMmotorstarter[7].et200SpMotorstarterOutputs[0..1].reserve10 := FALSE;
   unitMotorstarter[0].EMmotorstarter[0].et200SpMotorstarterOutputs[0..1].disableQuickStop := FALSE;
   unitMotorstarter[0].EMmotorstarter[1].et200SpMotorstarterOutputs[0..1].disableQuickStop := FALSE;
   unitMotorstarter[0].EMmotorstarter[2].et200SpMotorstarterOutputs[0..1].disableQuickStop := FALSE;
   unitMotorstarter[0].EMmotorstarter[3].et200SpMotorstarterOutputs[0..1].disableQuickStop := FALSE;
   unitMotorstarter[0].EMmotorstarter[4].et200SpMotorstarterOutputs[0..1].disableQuickStop := FALSE;
   unitMotorstarter[0].EMmotorstarter[5].et200SpMotorstarterOutputs[0..1].disableQuickStop := FALSE;
   unitMotorstarter[0].EMmotorstarter[6].et200SpMotorstarterOutputs[0..1].disableQuickStop := FALSE;
   unitMotorstarter[0].EMmotorstarter[7].et200SpMotorstarterOutputs[0..1].disableQuickStop := FALSE;
END_DATA_BLOCK
